{attribute 'qualified_only'}
{attribute 'strict'}
TYPE L_Stopper :
(
	ST1 := 1,
    ST2 := 2
);
END_TYPE

(* stored: Version 1.1.0.1, ProductVersion 3.1.4022.18
   EnumerationTextList L_Stopper: Id {e3c9e6c4-2110-466d-b87d-181f146f8f2a} *)
